// 40 Visualizations/COLLECTOR/VIS_SENSOR_COLLECTOR_TEMP
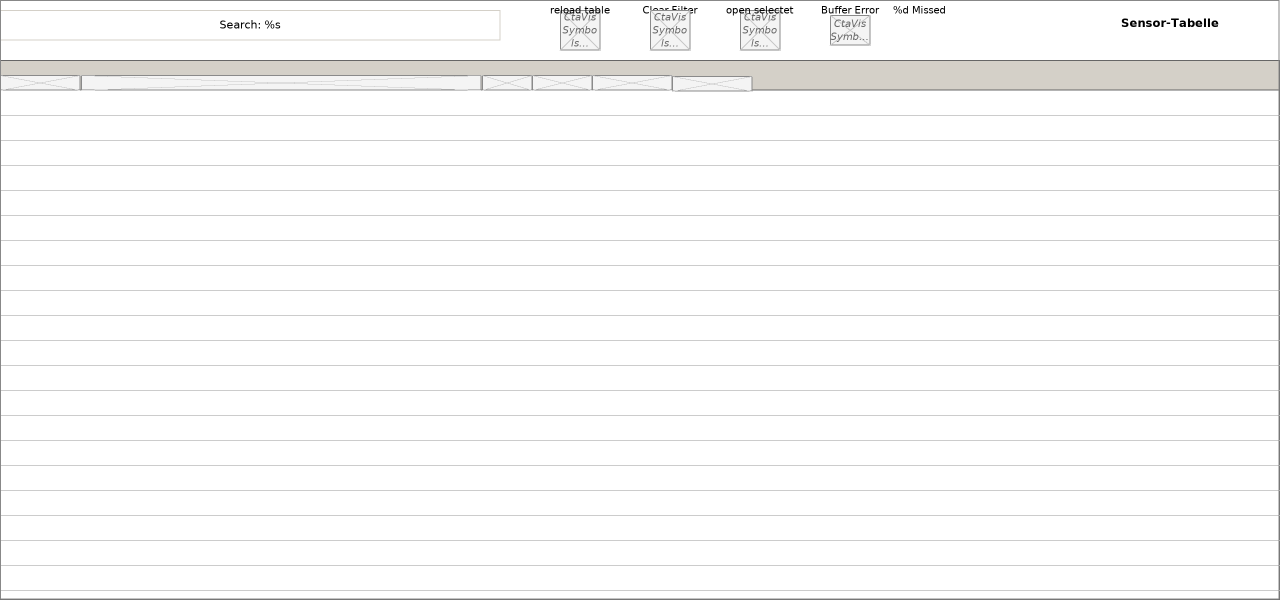
VISUALIZATION VIS_SENSOR_COLLECTOR_TEMP  // 1280x600
VAR_INPUT
	aySensorTabellenInfo   : ARRAY[1..Parameter.iMaxSensor] OF ITF_SENSOR_TABELLE_INFO;
    uiMax                   : UINT;
    ITF_SENSOR_COLLECTOR   : ITF_SENSOR_COLLECTOR;
END_VAR
VAR
    iZeile                  :   INT;
    stSearch                :   STRING;
    uiSort                  :   UINT;
    xReadySearch            :   BOOL;
END_VAR
    Table (0,60 1280x540), data array: aySensorTabellenInfo
        p1128707560: uiMax
        p1014161805: Parameter.iMaxSensor - 1 + 1
        p1137915858: iZeile
        p1933151965: aySensorTabellenInfo[INDEX].proNoBmkInList
        p3863566920: aySensorTabellenInfo[INDEX].proGetInstancePath
        p2192122294: aySensorTabellenInfo[INDEX].proSetInstancePath
        p3854506369: aySensorTabellenInfo[INDEX].proGetBMK
        p516019884: aySensorTabellenInfo[INDEX].proGetObjectId
        p2243050616: aySensorTabellenInfo[INDEX].proGetCustomerDesignation
        p4088588272: aySensorTabellenInfo[INDEX].proGetAKS
        p1892666644: aySensorTabellenInfo[INDEX].proGetVendorDesignation
        p511219082: Vendor designation
        p1757482276: Value OUT
        p746581629: aySensorTabellenInfo[INDEX].proSoftwareValue
        p4092479075: Enabled
        p2170511999: aySensorTabellenInfo[INDEX].proEnSymbol
        p338671338: aySensorTabellenInfo[INDEX].proStateSymbol
        p1218418051: aySensorTabellenInfo[INDEX].proRawValue
        p505689113: Value IN
        p3723444502: aySensorTabellenInfo[INDEX].proPhysicalValue
        p2237128397: Physical IN
    Image (740,10 40x40), invisible if: TO_DINT(iZeile) < LOWER_BOUND(aySensorTabellenInfo,1) OR TO_DINT(iZeile) > UPPER_BOUND(aySensorTabellenInfo,1), image: CtaVisSymbols.ImagePool.Sensor_Black
        OnMouseClick:  Dialog=POPUP_SENSOR, Parameters={uiPopUpGruppe: 0, ITF_SENSORIN: ITF_SENSOR_COLLECTOR.metGetAntriebITF(iZeile)}, OpenModal=True, OpenCentered=True
    Textfield (0,10 500x30), "Search: %s", text variable: stSearch
        OnMouseClick: write the text variable via Default
        OnMouseClick: execute { xReadySearch := TRUE; }
    Image (560,10 40x40), invisible if: NOT xReadySearch, image: CtaVisSymbols.ImagePool.refresh_solo_black
        OnMouseClick: execute { ITF_SENSOR_COLLECTOR.metSortArray(stSearch,uiSort); xReadySearch := FALSE; }
    Label (540,5 80x10), "reload table", invisible if: NOT xReadySearch
    Label (720,5 80x10), "open selectet", invisible if: TO_DINT(iZeile) < LOWER_BOUND(aySensorTabellenInfo,1) OR TO_DINT(iZeile) > UPPER_BOUND(aySensorTabellenInfo,1)
    Label (630,5 80x10), "Clear Filter", invisible if: stSearch = '' AND uiSort = 0
    Image (650,10 40x40), invisible if: stSearch = '' AND uiSort = 0, image: CtaVisSymbols.ImagePool.close_solo_black
        OnMouseClick: execute {
            stSearch := '';
            uiSort   := 0;
            ITF_SENSOR_COLLECTOR.metSortArray(stSearch,uiSort);
            xReadySearch := FALSE;
        }
    Label (1095,8 150x30), "Sensor-Tabelle"
    Label (810,5 80x10), "Buffer Error", invisible if: NOT ITF_SENSOR_COLLECTOR.proBufferError
    Image (830,15 40x30), invisible if: NOT ITF_SENSOR_COLLECTOR.proBufferError, image: CtaVisSymbols.ImagePool.CtaError
    Textfield (890,5 100x10), "%d Missed", text variable: ITF_SENSOR_COLLECTOR.proMissedBuffer, invisible if: NOT ITF_SENSOR_COLLECTOR.proBufferError
    Frame (672,61 80x30)
        shows SelSort(uiSel := uiSort, stSearch := stSearch, ITF_SENSOR_COLLECTOR := ITF_SENSOR_COLLECTOR, uiValue := 6)
    Frame (592,60 80x30)
        shows SelSort(uiSel := uiSort, stSearch := stSearch, ITF_SENSOR_COLLECTOR := ITF_SENSOR_COLLECTOR, uiValue := 5)
    Frame (532,60 60x30)
        shows SelSort(uiSel := uiSort, stSearch := stSearch, ITF_SENSOR_COLLECTOR := ITF_SENSOR_COLLECTOR, uiValue := 4)
    Frame (482,60 50x30)
        shows SelSort(uiSel := uiSort, stSearch := stSearch, ITF_SENSOR_COLLECTOR := ITF_SENSOR_COLLECTOR, uiValue := 3)
    Frame (81,60 400x30)
        shows SelSort(uiSel := uiSort, stSearch := stSearch, ITF_SENSOR_COLLECTOR := ITF_SENSOR_COLLECTOR, uiValue := 2)
    Frame (0,60 80x30)
        shows SelSort(uiSel := uiSort, stSearch := stSearch, ITF_SENSOR_COLLECTOR := ITF_SENSOR_COLLECTOR, uiValue := 1)
END_VISUALIZATION

// 40 Visualizations/COLLECTOR/Help Funktionen/SortPfeil
VISUALIZATION SortPfeil  // 15x15
    Image (0,0 15x15), image: CtaVisSymbols.ImagePool.arrow-down_solo_black
END_VISUALIZATION

// 40 Visualizations/POPUP/POPUP_SENSOR
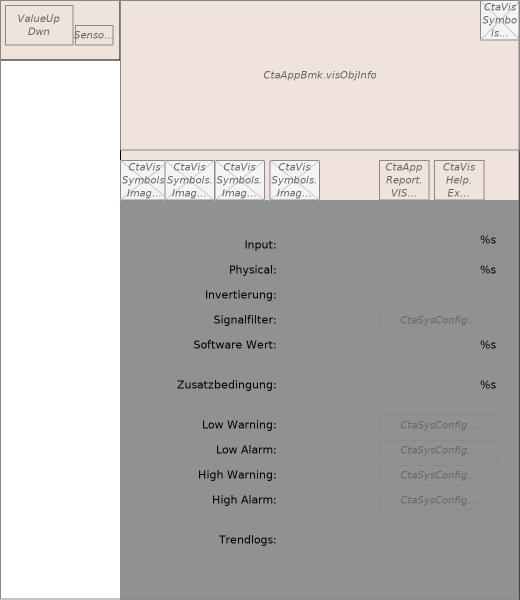
VISUALIZATION POPUP_SENSOR  // 520x600
VAR_INPUT
	ITF_SENSORIN	:	ITF_SENSOR;
	stExklParameter	:	STRING [40];
	uiPopUpGruppe 	: 	UINT;
END_VAR
    Rectangle (0,0 120x60)
    Rectangle (120,0 400x600)
    Frame (120,0 400x150)
        shows CtaAppBmk.visObjInfo(ITF_BMK_IN := ITF_SENSORIN)
    Image (480,0 40x40), image: CtaVisSymbols.ImagePool.close_solo_black
        OnMouseClick:  Dialog=POPUP_SENSOR, Result=None, NumpadKeypadSet=True
    Frame (120,200 399x400), frame switch variable: uiPopUpGruppe
        shows VIS_SENSOR_OVERVIEW(ITF_SENSORIN := ITF_SENSORIN)
        shows VIS_SENSOR_MANUAL(ITF_SENSORIN := ITF_SENSORIN)
        shows VIS_SENSOR_PARAMETER(ITF_SENSORIN := ITF_SENSORIN)
        shows Sensor_BUS(ITF_SENSORIN := ITF_SENSORIN)
        shows VIS_SENSOR_REPORTS(ITF_SENSORIN := ITF_SENSORIN)
        shows VIS_ANTRIEB_REPORTS(ITF_SENSORIN := ITF_SENSOR_IN)
    Frame (120,160 399x40)
        shows VIS_SENSOR_LISTE(uiPopUpGruppe := uiPopUpGruppe, xHand := ITF_SENSORIN.proIsHandOnOrOff, xHandOff := ITF_SENSORIN.proHandOff, ITF_REPORTMANAGER_IN := ITF_SENSORIN.proITF_REPORTMANAGER, stExklParameter := stExklParameter)
        pReferences[0]: AnzError=ITF_SENSORIN.proCountedError, AnzWarning=ITF_SENSORIN.proCountedWarning
    Frame (5,5 110x50), input disabled if: TRUE, frame switch variable: ITF_SENSORIN.proAtIconNr
        shows VIS_SENSOR_FLAT_LEFT_ABOVE(ITF_SENSOR_IN := ITF_SENSORIN, stExklParameter := stExklParameter)
        shows VIS_SENSOR_FLAT_LEFT_BELOW(ITF_SENSOR_IN := ITF_SENSORIN, stExklParameter := stExklParameter)
        shows VIS_SENSOR_FLAT_RIGHT_ABOVE(ITF_SENSOR_IN := ITF_SENSORIN, stExklParameter := stExklParameter)
        shows VIS_SENSOR_FLAT_RIGHT_BELOW(ITF_SENSOR_IN := ITF_SENSORIN, stExklParameter := stExklParameter)
        shows VIS_SENSOR_ROUND_RIGHT_ABOVE(ITF_SENSOR_IN := ITF_SENSORIN, stExklParameter := stExklParameter)
        shows VIS_SENSOR_ROUND_RIGHT_BELOW(ITF_SENSOR_IN := ITF_SENSORIN, stExklParameter := stExklParameter)
        shows VIS_SENSOR_ROUND_LEFT_ABOVE(ITF_SENSOR_IN := ITF_SENSORIN, stExklParameter := stExklParameter)
        shows VIS_SENSOR_ROUND_LEFT_BELOW(ITF_SENSOR_IN := ITF_SENSORIN, stExklParameter := stExklParameter)
END_VISUALIZATION

// 40 Visualizations/POPUP/VIS_SENSOR_LISTE
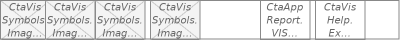
VISUALIZATION VIS_SENSOR_LISTE  // 400x40
VAR_IN_OUT
	uiPopUpGruppe : UINT;
END_VAR
VAR_INPUT
    xHand           		: BOOL;
    xHandOff        		: BOOL;
    ITF_REPORTMANAGER_IN    : CtaAppReport.ITF_REPORTMANAGER;
	stExklParameter			: STRING [40];
END_VAR
    Rectangle (5,0 40x40), colour toggle: uiPopUpGruppe = 0
        OnMouseDown: execute { uiPopUpGruppe := 0; }
    Image (0,0 50x40), image: CtaVisSymbols.ImagePool.eye
        OnMouseDown: execute { uiPopUpGruppe := 0; }
    Rectangle (50,0 40x40), colour toggle: uiPopUpGruppe = 1
        OnMouseDown: execute { uiPopUpGruppe := 1; }
    Image (45,0 50x40), invisible if: NOT xHand, image: CtaVisSymbols.ImagePool.front_hand_Yellow
        OnMouseDown: execute { uiPopUpGruppe := 1; }
    Image (45,0 50x40), image: CtaVisSymbols.ImagePool.front_hand_Black
        OnMouseDown: execute { uiPopUpGruppe := 1; }
    Image (45,0 50x40), invisible if: NOT xHandOff, image: CtaVisSymbols.ImagePool.front_hand_Yellow_Off
        OnMouseDown: execute { uiPopUpGruppe := 1; }
    Rectangle (100,0 40x40), colour toggle: uiPopUpGruppe = 2
        OnMouseDown: execute { uiPopUpGruppe := 2; }
    Image (95,0 50x40), image: CtaVisSymbols.ImagePool.gear
        OnMouseDown: execute { uiPopUpGruppe := 2; }
    Rectangle (155,0 40x40), colour toggle: uiPopUpGruppe = 3
        OnMouseDown: execute { uiPopUpGruppe := 3; }
    Image (150,0 50x40), image: CtaVisSymbols.ImagePool.lan
        OnMouseDown: execute { uiPopUpGruppe := 3; }
    Rectangle (265,0 40x40), colour toggle: uiPopUpGruppe = 4
        OnMouseDown: execute { uiPopUpGruppe := 4; }
    Frame (260,0 50x40)
        shows CtaAppReport.VIS_ANZ_REPORTS_MODUL(ITF_REPORTMANAGER_IN := ITF_REPORTMANAGER_IN)
        OnMouseClick: execute { uiPopUpGruppe := 4; }
    Rectangle (320,0 40x40)
    Frame (315,0 50x40)
        shows CtaVisHelp.ExkParameterSymbol(stExklParameter := stExklParameter)
END_VISUALIZATION

// 40 Visualizations/POPUP/PARAMETER/SENSOR_ReportManagement/Sensor_LowAlarm_Param
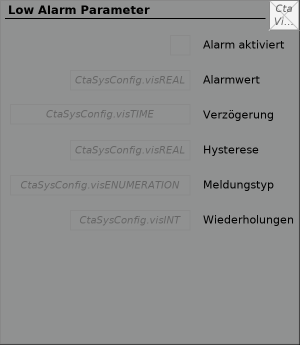
VISUALIZATION Sensor_LowAlarm_Param  // 300x345
VAR_INPUT
	ITF_SENSORIN	:	ITF_SENSOR;
END_VAR
VAR_IN_OUT
    xShow   :   BOOL;
END_VAR
    Rectangle (0,0 300x345)
    Image (269,0 30x30), image: CtaVisSymbols.ImagePool.close_solo_black
        OnMouseClick: execute { xShow := FALSE; }
    Label (5,0 198x20), "Low Alarm Parameter"
    Line (5,18) (265,18)
    Label (200,35 100x20), "Alarm aktiviert"
    Frame (170,35 20x20)
        shows CtaSysConfig.visBOOL(visfbBOOLIn := ITF_SENSORIN.P_scLoAlarm_fbxDoesAlarm)
    Label (200,70 100x20), "Alarmwert"
    Frame (70,70 120x20), invisible if: (ITF_SENSORIN.proValueInputType = enInputType.DigitalInput) OR (ITF_SENSORIN.proValueInputType = enInputType.Digital_ITF_Input)
        shows CtaSysConfig.visREAL(visfbREALIn := ITF_SENSORIN.P_scLoAlarm_fbrValue)
    Label (200,105 100x20), "Verzögerung"
    Frame (10,104 180x20)
        shows CtaSysConfig.visTIME(visfbTIMEIn := ITF_SENSORIN.P_scLoAlarm_fbtDelayTillAlarm)
    Frame (70,140 120x20), invisible if: (ITF_SENSORIN.proValueInputType = enInputType.DigitalInput) OR (ITF_SENSORIN.proValueInputType = enInputType.Digital_ITF_Input)
        shows CtaSysConfig.visREAL(visfbREALIn := ITF_SENSORIN.P_scLoAlarm_fbrHysterese)
    Label (200,140 100x20), "Hysterese"
    Frame (10,175 180x20), text list: 'CtaAppReport.txtLibAp99_2enTypeOfAck', text index: CtaSysConfig.fcGetEnumerationId(ITF_SENSORIN.P_scLoAlarm_fbiTypeOfAcknolage)
        shows CtaSysConfig.visENUMERATION(visfbENUIn := ITF_SENSORIN.P_scLoAlarm_fbiTypeOfAcknolage)
    Label (200,175 100x20), "Meldungstyp"
    Frame (70,210 120x20), invisible if: NOT (CtaSysConfig.fcGetEnumerationId(ITF_SENSORIN.P_scLoAlarm_fbiTypeOfAcknolage) = 2)
        shows CtaSysConfig.visINT(visfbINTIn := ITF_SENSORIN.P_scLoAlarm_fbiRetryTillLock)
    Label (200,210 100x20), "Wiederholungen"
END_VISUALIZATION

// 40 Visualizations/ICON/SENSOR_FLAT/SENSOR_FLAT_TXT_LEFT/ABOVE/VIS_SENSOR_FLAT_LeftAboveCheckQuerry
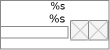
VISUALIZATION VIS_SENSOR_FLAT_LeftAboveCheckQuerry  // 110x50
VAR_INPUT
    ITF_SENSOR_IN   :   ITF_SENSOR;
	stExklParameter	:	STRING [40];	
END_VAR
    Frame (0,0 110x50)
        shows VIS_SENSOR_FLAT_LeftAboveCheckIsEnabled(ITF_SENSOR_IN := ITF_SENSOR_IN, stExklParameter := stExklParameter)
END_VISUALIZATION

// 40 Visualizations/ICON/SENSOR_FLAT/SENSOR_FLAT_TXT_LEFT/ABOVE/VIS_SENSOR_FLAT_LEFT_ABOVE
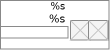
VISUALIZATION VIS_SENSOR_FLAT_LEFT_ABOVE  // 110x50
VAR_INPUT
    ITF_SENSOR_IN   :   ITF_SENSOR;	
END_VAR
VAR_INPUT CONSTANT	
	stExklParameter	:	STRING [40] := ' ';	
END_VAR
VAR CONSTANT
	uiIconNr		: UINT := 0;
END_VAR
    Frame (0,0 110x50), invisible if: NOT fcCheckQuerryAndIconReturn(_ITF_IN := ITF_SENSOR_IN, _uiIconNr_IN := uiIconNr)
        shows VIS_SENSOR_FLAT_LeftAboveCheckQuerry(ITF_SENSOR_IN := ITF_SENSOR_IN, stExklParameter := stExklParameter)
END_VISUALIZATION

// 40 Visualizations/ICON/SENSOR_FLAT/SENSOR_FLAT_TXT_LEFT/ABOVE/VIS_SENSOR_FLAT_LeftAboveCheckIsEnabled
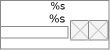
VISUALIZATION VIS_SENSOR_FLAT_LeftAboveCheckIsEnabled  // 110x50
VAR_INPUT
    ITF_SENSOR_IN   :   ITF_SENSOR;
	stExklParameter	:	STRING [40];	
END_VAR
    Frame (70,20 38x20), invisible if: NOT ITF_SENSOR_IN.proIsEnabled
        shows SensorFlat(ITF_SENSORIN := ITF_SENSOR_IN)
    Frame (0,0 68x40), invisible if: NOT ITF_SENSOR_IN.proIsEnabled
        shows ValueUpDwn(ITF_SENSORIN := ITF_SENSOR_IN, uiTextAusrichtung := 6)
    Rectangle (0,0 110x50)
        OnMouseClick:  Dialog=POPUP_SENSOR, Parameters={stExklParameter: stExklParameter, ITF_SENSORIN: ITF_SENSOR_IN, uiPopUpGruppe: 0}, OpenCentered=True
END_VISUALIZATION

// 40 Visualizations/ICON/SENSOR_FLAT/SENSOR_FLAT_TXT_RIGHT/ABOVE/VIS_SENSOR_FLAT_RigthAboveCheckIsEnabled
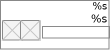
VISUALIZATION VIS_SENSOR_FLAT_RigthAboveCheckIsEnabled  // 110x50
VAR_INPUT
    ITF_SENSOR_IN   :   ITF_SENSOR;
	stExklParameter	:	STRING [40];	
END_VAR
    Frame (2,20 38x20), invisible if: NOT ITF_SENSOR_IN.proIsEnabled
        shows SensorFlat(ITF_SENSORIN := ITF_SENSOR_IN)
    Frame (42,0 68x40), invisible if: NOT ITF_SENSOR_IN.proIsEnabled
        shows ValueUpDwn(ITF_SENSORIN := ITF_SENSOR_IN, uiTextAusrichtung := 4)
    Rectangle (0,0 110x50)
        OnMouseClick:  Dialog=POPUP_SENSOR, Parameters={stExklParameter: stExklParameter, ITF_SENSORIN: ITF_SENSOR_IN, uiPopUpGruppe: 0}, OpenCentered=True
END_VISUALIZATION

// 40 Visualizations/ICON/SENSOR_BASE/ICON/Flat/SensorFlat
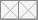
VISUALIZATION SensorFlat  // 38x20
VAR_INPUT
    ITF_SENSORIN   :   ITF_SENSOR;	
END_VAR
    RoundedRectangle (0,0 38x20), colour toggle: ITF_SENSORIN.proAcknowlege, invisible if: ITF_SENSORIN.proIsError
    RoundedRectangle (0,0 38x20), colour toggle: ITF_SENSORIN.proIsError
    Image (0,0 20x20), invisible if: NOT ITF_SENSORIN.proIsWarning, image: CtaVisSymbols.ImagePool.CtaWarning
    Image (18,0 20x20), invisible if: NOT ITF_SENSORIN.proIsHandOnOrOff, image: CtaVisSymbols.ImagePool.front_hand_Yellow
    Image (18,0 20x20), invisible if: NOT ITF_SENSORIN.proHandOff, image: CtaVisSymbols.ImagePool.front_hand_Yellow_Off
END_VISUALIZATION

// 40 Visualizations/POPUP/PARAMETER/VIS_SENSOR_PARAMETER
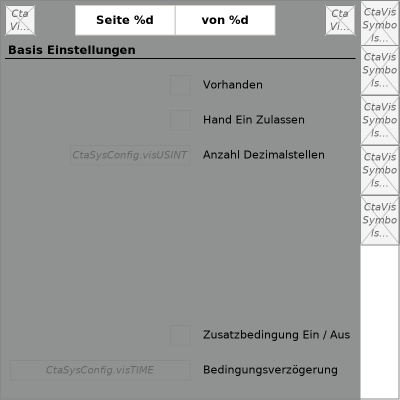
VISUALIZATION VIS_SENSOR_PARAMETER  // 400x400
VAR_INPUT
    ITF_SENSORIN : ITF_SENSOR;
END_VAR
VAR
    uiParameterGruppe : UINT;
END_VAR
    Image (145,122 150x30), image: ImagePool.Kreis
    Frame (360,0 40x300)
        shows VIS_SENSOR_PARAMETER_LISTE(enValueInputType := ITF_SENSORIN.proValueInputType, uiParameterGruppe := uiParameterGruppe)
    Frame (0,0 360x400), frame switch variable: uiParameterGruppe
        shows VIS_SENSOR_PARAMETER_BASE(ITF_SENSORIN := ITF_SENSORIN)
        shows VIS_SENSOR_PARAMETER_FILTER(ITF_SENSORIN := ITF_SENSORIN)
        shows VIS_SENSOR_PARAMETER_REPORTMNG(ITF_SENSORIN := ITF_SENSORIN)
        shows VIS_SENSOR_IO_PARAMETER(ITF_SENSORIN := ITF_SENSORIN)
        shows VIS_SENSOR_PARAMETER_TRENDLOG(ITF_SENSORIN := ITF_SENSORIN)
        pReferences[3]: ITF_IO_IN=ITF_SENSOR_IN.proIO_ITF
END_VISUALIZATION

// 40 Visualizations/POPUP/PARAMETER/VIS_SENSOR_PARAMETER_LISTE
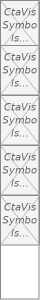
VISUALIZATION VIS_SENSOR_PARAMETER_LISTE  // 40x300
VAR_INPUT
	enValueInputType : enInputType;
END_VAR
VAR_IN_OUT
	uiParameterGruppe : UINT;
END_VAR
    Rectangle (0,5 39x40), colour toggle: uiParameterGruppe = 0
        OnMouseDown: execute { uiParameterGruppe := 0; }
    Image (0,0 40x50), image: CtaVisSymbols.ImagePool.Sensor_Black
        OnMouseDown: execute { uiParameterGruppe := 0; }
    Rectangle (0,50 39x40), colour toggle: uiParameterGruppe = 1
        OnMouseDown: execute { uiParameterGruppe := 1; }
    Image (0,45 40x50), image: CtaVisSymbols.ImagePool.SearchFilter
        OnMouseDown: execute { uiParameterGruppe := 1; }
    Rectangle (0,100 39x40), colour toggle: uiParameterGruppe = 2
        OnMouseDown: execute { uiParameterGruppe := 2; }
    Image (0,95 40x50), image: CtaVisSymbols.ImagePool.notification_black
        OnMouseDown: execute { uiParameterGruppe := 2; }
    Rectangle (1,150 39x40), colour toggle: uiParameterGruppe = 3, invisible if: enValueInputType = 0 OR enValueInputType = 1 OR enValueInputType = 2, input disabled if: enValueInputType = 0 OR enValueInputType = 1 OR enValueInputType = 2
        OnMouseDown: execute { uiParameterGruppe := 3; }
    Image (0,145 40x50), invisible if: enValueInputType = 0 OR enValueInputType = 1 OR enValueInputType = 2, input disabled if: enValueInputType = 0 OR enValueInputType = 1 OR enValueInputType = 2, image: CtaVisSymbols.ImagePool.dip-switch
        OnMouseDown: execute { uiParameterGruppe := 3; }
    Rectangle (0,200 39x40), colour toggle: uiParameterGruppe = 4
        OnMouseDown: execute { uiParameterGruppe := 4; }
    Image (0,195 40x50), image: CtaVisSymbols.ImagePool.sine-wave
        OnMouseDown: execute { uiParameterGruppe := 4; }
END_VISUALIZATION

// 40 Visualizations/POPUP/MANUAL/VIS_SENSOR_MANUAL
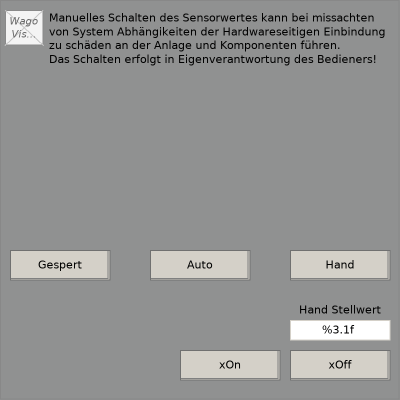
VISUALIZATION VIS_SENSOR_MANUAL  // 400x400
VAR_INPUT
    ITF_SENSORIN    :   ITF_SENSOR;	
END_VAR
    Button (10,250 100x30), "Gespert", colour toggle: ITF_SENSORIN.proHandOff, pressed state: ITF_SENSORIN.proHandOff
        toggle ITF_SENSORIN.proHandOff
    Button (290,250 100x30), "Hand", colour toggle: ITF_SENSORIN.proHandOn, pressed state: ITF_SENSORIN.proHandOn
        toggle ITF_SENSORIN.proHandOn
    Button (150,250 100x30), "Auto", colour toggle: ITF_SENSORIN.proAuto, pressed state: ITF_SENSORIN.proAuto
        toggle ITF_SENSORIN.proAuto
    Label (46,10 350x100), "Manuelles Schalten des Sensorwertes kann bei missachten von System Abhängikeiten der Hardwareseitigen Einbindung zu schäden an der Anlage und Komponenten führen. Das Schalten erfolgt in Eigenverantwortung des Bedieners!"
    Textfield (290,320 100x20), "%3.1f", text variable: ITF_SENSORIN.proHandOnY, invisible if: ITF_SENSORIN.proValueInputType = 0 OR ITF_SENSORIN.proValueInputType = 2 OR ITF_SENSORIN.proValueInputType = 4
        OnMouseClick: write the text variable via InputWithLimits, min 0, max 100, title 'Stellwert'
    Image (5,10 38x35), image: WagoVisuIcons.WagoIcons.2
    Label (290,300 100x20), "Hand Stellwert"
    Button (290,350 100x30), "xOff", colour toggle: ITF_SENSORIN.proManualFalse, pressed state: ITF_SENSORIN.proManualFalse, invisible if: ITF_SENSORIN.proValueInputType = 0 OR ITF_SENSORIN.proValueInputType = 1 OR ITF_SENSORIN.proValueInputType = 3
        toggle ITF_SENSORIN.proManualFalse
    Button (180,350 100x30), "xOn", colour toggle: ITF_SENSORIN.proManualTrue, pressed state: ITF_SENSORIN.proManualTrue, invisible if: ITF_SENSORIN.proValueInputType = 0 OR ITF_SENSORIN.proValueInputType = 1 OR ITF_SENSORIN.proValueInputType = 3
        toggle ITF_SENSORIN.proManualTrue
END_VISUALIZATION

// 40 Visualizations/POPUP/OVERVIEW/VIS_SENSOR_OVERVIEW
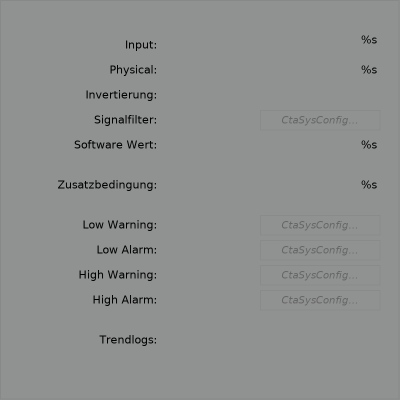
VISUALIZATION VIS_SENSOR_OVERVIEW  // 400x400
VAR_INPUT
    ITF_SENSORIN	:	ITF_SENSOR;
END_VAR
    Frame (0,0 400x400), invisible if: NOT __QUERYINTERFACE(ITF_SENSORIN,ITF_SENSORIN)
        shows VIS_SENSOR_OVERVIEW0(ITF_SENSORIN := ITF_SENSORIN)
END_VISUALIZATION

// 40 Visualizations/POPUP/PARAMETER/SENSOR_ReportManagement/Sensor_HighAlarm_Param
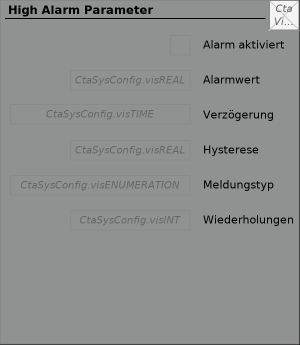
VISUALIZATION Sensor_HighAlarm_Param  // 300x345
VAR_INPUT
	ITF_SENSORIN	:	ITF_SENSOR;
END_VAR
VAR_IN_OUT
    xShow   :   BOOL;
END_VAR
    Rectangle (0,0 300x345)
    Image (269,0 30x30), image: CtaVisSymbols.ImagePool.close_solo_black
        OnMouseClick: execute { xShow := FALSE; }
    Label (5,0 198x20), "High Alarm Parameter"
    Line (5,18) (265,18)
    Label (200,35 100x20), "Alarm aktiviert"
    Frame (170,35 20x20)
        shows CtaSysConfig.visBOOL(visfbBOOLIn := ITF_SENSORIN.P_scHighAlram_fbxDoesAlarm)
    Label (200,70 100x20), "Alarmwert"
    Frame (70,70 120x20), invisible if: (ITF_SENSORIN.proValueInputType = enInputType.DigitalInput) OR (ITF_SENSORIN.proValueInputType = enInputType.Digital_ITF_Input)
        shows CtaSysConfig.visREAL(visfbREALIn := ITF_SENSORIN.P_scHighAlarm_fbrValue)
    Label (200,105 100x20), "Verzögerung"
    Frame (10,104 180x20)
        shows CtaSysConfig.visTIME(visfbTIMEIn := ITF_SENSORIN.P_scHighAlarm_fbtDelayTillAlarm)
    Frame (70,140 120x20), invisible if: (ITF_SENSORIN.proValueInputType = enInputType.DigitalInput) OR (ITF_SENSORIN.proValueInputType = enInputType.Digital_ITF_Input)
        shows CtaSysConfig.visREAL(visfbREALIn := ITF_SENSORIN.P_scHighAlarm_fbrHysterese)
    Label (200,140 100x20), "Hysterese"
    Frame (10,175 180x20), text list: 'CtaAppReport.txtLibAp99_2enTypeOfAck', text index: CtaSysConfig.fcGetEnumerationId(ITF_SENSORIN.P_scHighAlarm_fbiTypeOfAcknolage)
        shows CtaSysConfig.visENUMERATION(visfbENUIn := ITF_SENSORIN.P_scHighAlarm_fbiTypeOfAcknolage)
    Label (200,175 100x20), "Meldungstyp"
    Frame (70,210 120x20), invisible if: NOT (CtaSysConfig.fcGetEnumerationId(ITF_SENSORIN.P_scHighAlarm_fbiTypeOfAcknolage) = 2)
        shows CtaSysConfig.visINT(visfbINTIn := ITF_SENSORIN.P_scHighAlarm_fbiRetryTillLock)
    Label (200,210 100x20), "Wiederholungen"
END_VISUALIZATION

// 40 Visualizations/ICON/SENSOR_FLAT/SENSOR_FLAT_TXT_LEFT/BELOW/VIS_SENSOR_FLAT_LEFT_BELOW
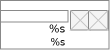
VISUALIZATION VIS_SENSOR_FLAT_LEFT_BELOW  // 110x50
VAR_INPUT
    ITF_SENSOR_IN   :   ITF_SENSOR;	
END_VAR
VAR_INPUT CONSTANT	
	stExklParameter	:	STRING [40] := ' ';	
END_VAR
VAR CONSTANT
	uiIconNr		: UINT := 1;
END_VAR
    Frame (0,0 110x50), invisible if: NOT fcCheckQuerryAndIconReturn(_ITF_IN := ITF_SENSOR_IN, _uiIconNr_IN := uiIconNr)
        shows VIS_SENSOR_FLAT_LeftBelowCheckQuerry(ITF_SENSOR_IN := ITF_SENSOR_IN, stExklParameter := stExklParameter)
END_VISUALIZATION

// 40 Visualizations/POPUP/PARAMETER/SENSOR_ReportManagement/Sensor_HighWarning_Param
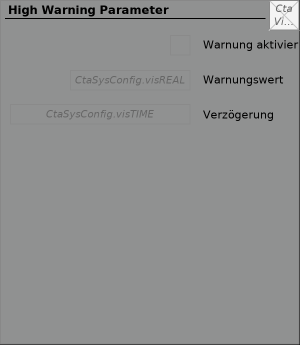
VISUALIZATION Sensor_HighWarning_Param  // 300x345
VAR_INPUT
	ITF_SENSORIN	:	ITF_SENSOR;
END_VAR
VAR_IN_OUT
    xShow   :   BOOL;
END_VAR
    Rectangle (0,0 300x345)
    Image (269,0 30x30), image: CtaVisSymbols.ImagePool.close_solo_black
        OnMouseClick: execute { xShow := FALSE; }
    Label (5,0 198x20), "High Warning Parameter"
    Line (5,18) (265,18)
    Label (200,35 100x20), "Warnung aktiviert"
    Frame (170,35 20x20)
        shows CtaSysConfig.visBOOL(visfbBOOLIn := ITF_SENSORIN.P_scHighWarning_fbxDoesWarning)
    Label (200,70 100x20), "Warnungswert"
    Frame (70,70 120x20), invisible if: (ITF_SENSORIN.proValueInputType = enInputType.DigitalInput) OR (ITF_SENSORIN.proValueInputType = enInputType.Digital_ITF_Input)
        shows CtaSysConfig.visREAL(visfbREALIn := ITF_SENSORIN.P_scHighWarning_fbrValue)
    Label (200,105 100x20), "Verzögerung"
    Frame (10,104 180x20)
        shows CtaSysConfig.visTIME(visfbTIMEIn := ITF_SENSORIN.P_scHighWarning_fbtDelayTillWarning)
END_VISUALIZATION

// 40 Visualizations/ICON/SENSOR_FLAT/SENSOR_FLAT_TXT_LEFT/BELOW/VIS_SENSOR_FLAT_LeftBelowCheckIsEnabled
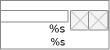
VISUALIZATION VIS_SENSOR_FLAT_LeftBelowCheckIsEnabled  // 110x50
VAR_INPUT
    ITF_SENSOR_IN   :   ITF_SENSOR;
	stExklParameter	:	STRING [40];	
END_VAR
    Frame (70,10 38x20), invisible if: NOT ITF_SENSOR_IN.proIsEnabled
        shows SensorFlat(ITF_SENSORIN := ITF_SENSOR_IN)
    Frame (0,10 68x40), invisible if: NOT ITF_SENSOR_IN.proIsEnabled
        shows ValueDwnUp(ITF_SENSORIN := ITF_SENSOR_IN, uiTextAusrichtung := 6)
    Rectangle (0,0 110x50)
        OnMouseClick:  Dialog=POPUP_SENSOR, Parameters={stExklParameter: stExklParameter, ITF_SENSORIN: ITF_SENSOR_IN, uiPopUpGruppe: 0}, OpenCentered=True
END_VISUALIZATION

// 40 Visualizations/POPUP/REPORTS/VIS_SENSOR_REPORTS
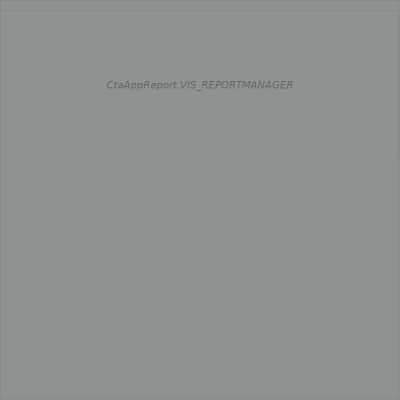
VISUALIZATION VIS_SENSOR_REPORTS  // 400x400
VAR_INPUT
    ITF_SENSORIN    :   ITF_SENSOR;	
END_VAR
    Frame (0,10 400x150)
        shows CtaAppReport.VIS_REPORTMANAGER(ITF_REPORTMANAGER := ITF_SENSORIN.proITF_REPORTMANAGER)
END_VISUALIZATION

// 40 Visualizations/POPUP/PARAMETER/SENSOR_ParameterBase/VIS_SENSOR_PARAMETER_BASE0
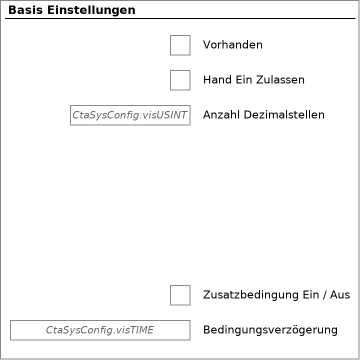
VISUALIZATION VIS_SENSOR_PARAMETER_BASE0  // 360x360
VAR_INPUT
    ITF_SENSORIN	:  ITF_SENSOR;
END_VAR
    Label (5,0 350x20), "Basis Einstellungen"
    Line (5,18) (355,18)
    Label (200,35 150x20), "Vorhanden"
    Label (200,70 150x20), "Hand Ein Zulassen"
    Frame (170,35 20x20)
        shows CtaSysConfig.visBOOL(visfbBOOLIn := ITF_SENSORIN.P_scBase_fbxEnable)
    Frame (170,70 20x20)
        shows CtaSysConfig.visBOOL(visfbBOOLIn := ITF_SENSORIN.P_scManual_fbxAllowManualOn)
    Frame (170,285 20x20)
        shows CtaSysConfig.visBOOL(visfbBOOLIn := ITF_SENSORIN.P_scAlCondition_fbxEnable)
    Label (200,285 150x20), "Zusatzbedingung Ein / Aus"
    Frame (10,320 180x20)
        shows CtaSysConfig.visTIME(visfbTIMEIn := ITF_SENSORIN.P_scAlCondition_fbtDelayTillCondition)
    Label (200,320 150x20), "Bedingungsverzögerung"
    Frame (70,105 120x20), invisible if: NOT (ITF_SENSORIN.proValueInputType = enInputType.AnalogInput or ITF_SENSORIN.proValueInputType = enInputType.Analog_ITF_Input)
        shows CtaSysConfig.visUSINT(visfbUSINTIn := ITF_SENSORIN.P_scVisu_fbusiDezimalPos)
    Label (200,105 150x20), "Anzahl Dezimalstellen", invisible if: NOT (ITF_SENSORIN.proValueInputType = enInputType.AnalogInput or ITF_SENSORIN.proValueInputType = enInputType.Analog_ITF_Input)
END_VISUALIZATION

// 40 Visualizations/POPUP/PARAMETER/SENSOR_ParameterBase/VIS_SENSOR_PARAMETER_BASE
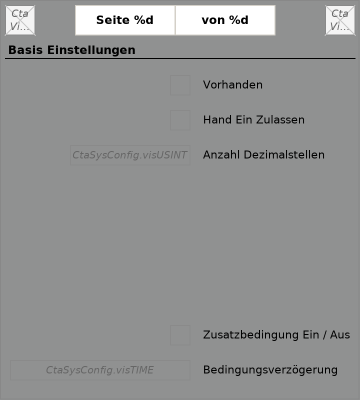
VISUALIZATION VIS_SENSOR_PARAMETER_BASE  // 360x400
VAR_INPUT
    ITF_SENSORIN 	: 	ITF_SENSOR;
END_VAR
VAR
    uiPage  :   UINT;
    uiMin   :   UINT    := 0;
    uiMax   :   UINT    := 0;
END_VAR
    Image (5,5 30x30), invisible if: uiPage = uiMin, image: CtaVisSymbols.ImagePool.arrow-left_square
        OnMouseClick: execute {
            uiPage := uiPage - 1;
            IF uiPage <= uiMin THEN
                uiPage := uiMin;
            END_IF;
        }
    Image (325,5 30x30), invisible if: uiPage = uiMax, image: CtaVisSymbols.ImagePool.arrow-right_square
        OnMouseClick: execute {
            uiPage := uiPage + 1;
            IF uiPage >= uiMax THEN
                uiPage := uiMax;
            END_IF;
        }
    Frame (0,40 360x360), frame switch variable: uiPage
        shows VIS_SENSOR_PARAMETER_BASE0(ITF_SENSORIN := ITF_SENSORIN)
        shows AT_ParameterIO1(ITF_Parameter := ITF_Parameter)
        pReferences[0]: ITF_Parameter=ITF_Parameter
    Textfield (175,5 100x30), "von %d", text variable: uiMax
    Textfield (75,5 100x30), "Seite %d", text variable: uiPage
END_VISUALIZATION

// 40 Visualizations/ICON/SENSOR_FLAT/SENSOR_FLAT_TXT_RIGHT/ABOVE/VIS_SENSOR_FLAT_RIGHT_ABOVE
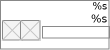
VISUALIZATION VIS_SENSOR_FLAT_RIGHT_ABOVE  // 110x50
VAR_INPUT
    ITF_SENSOR_IN   :   ITF_SENSOR;	
END_VAR
VAR_INPUT CONSTANT	
	stExklParameter	:	STRING [40] := ' ';	
END_VAR
VAR CONSTANT
	uiIconNr		:	UINT := 2;
END_VAR
    Frame (0,0 110x50), invisible if: NOT fcCheckQuerryAndIconReturn(_ITF_IN := ITF_SENSOR_IN, _uiIconNr_IN := uiIconNr)
        shows VIS_SENSOR_FLAT_RigthAboveCheckQuerry(ITF_SENSOR_IN := ITF_SENSOR_IN, stExklParameter := stExklParameter)
END_VISUALIZATION

// 40 Visualizations/ICON/SENSOR_FLAT/SENSOR_FLAT_TXT_LEFT/BELOW/VIS_SENSOR_FLAT_LeftBelowCheckQuerry
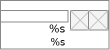
VISUALIZATION VIS_SENSOR_FLAT_LeftBelowCheckQuerry  // 110x50
VAR_INPUT
    ITF_SENSOR_IN   :   ITF_SENSOR;
	stExklParameter	:	STRING [40];	
END_VAR
    Frame (0,0 110x50)
        shows VIS_SENSOR_FLAT_LeftBelowCheckIsEnabled(ITF_SENSOR_IN := ITF_SENSOR_IN, stExklParameter := stExklParameter)
END_VISUALIZATION

// 40 Visualizations/POPUP/PARAMETER/SENSOR_ReportManagement/VIS_SENSOR_PARAMETER_REPORTMNG
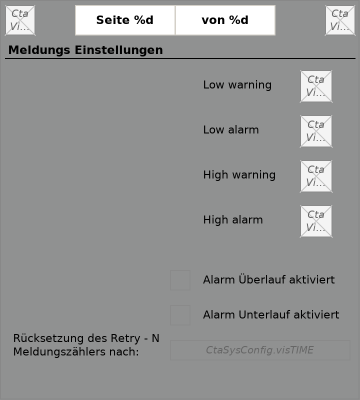
VISUALIZATION VIS_SENSOR_PARAMETER_REPORTMNG  // 360x400
VAR_INPUT
   	ITF_SENSORIN	:	ITF_SENSOR;
END_VAR
VAR
    uiPage  :   UINT;
    uiMin   :   UINT    := 0;
    uiMax   :   UINT    := 0;
END_VAR
    Image (5,5 30x30), invisible if: uiPage = uiMin, image: CtaVisSymbols.ImagePool.arrow-left_square
        OnMouseClick: execute {
            uiPage := uiPage - 1;
            IF uiPage <= uiMin THEN
                uiPage := uiMin;
            END_IF;
        }
    Image (325,5 30x30), invisible if: uiPage = uiMax, image: CtaVisSymbols.ImagePool.arrow-right_square
        OnMouseClick: execute {
            uiPage := uiPage + 1;
            IF uiPage >= uiMax THEN
                uiPage := uiMax;
            END_IF;
        }
    Frame (0,40 360x360), frame switch variable: uiPage
        shows VIS_SENSOR_PARAMETER_REPORTMNG_1(ITF_SENSORIN := ITF_SENSORIN)
        shows AT_ParameterIO1(ITF_Parameter := ITF_Parameter)
    Textfield (175,5 100x30), "von %d", text variable: uiMax
    Textfield (75,5 100x30), "Seite %d", text variable: uiPage
END_VISUALIZATION

// 40 Visualizations/POPUP/PARAMETER/SENSOR_ReportManagement/VIS_SENSOR_PARAMETER_REPORTMNG_1
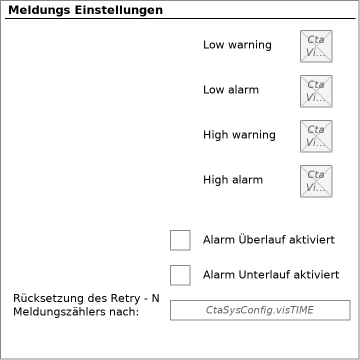
VISUALIZATION VIS_SENSOR_PARAMETER_REPORTMNG_1  // 360x360
VAR_INPUT
   	ITF_SENSORIN	:	ITF_SENSOR;
END_VAR
VAR
	xShowLoWarning	:	BOOL;
	xShowLoAlarm	:	BOOL;
	xShowHiWarning	:	BOOL;
	xShowHiAlarm	:	BOOL;
END_VAR
    Label (5,0 350x20), "Meldungs Einstellungen"
    Line (5,18) (355,18)
    Label (200,35 150x20), "Low warning"
    Label (200,80 150x20), "Low alarm"
    Label (200,125 150x20), "High warning"
    Label (200,170 150x20), "High alarm"
    Image (300,30 32x32), image: CtaVisSymbols. ImagePool.CtaInfo
        OnMouseClick: execute {
            xShowLoWarning	:=	TRUE;
            xShowLoAlarm	:=	FALSE;
            xShowHiWarning	:=	FALSE;
            xShowHiAlarm	:=	FALSE;
        }
    Frame (400,18 300x345), invisible if: NOT xShowLoWarning
        shows Sensor_LowWarning_Param(ITF_SENSORIN := ITF_SENSORIN, xShow := xShowLoWarning)
    Image (300,75 32x32), image: CtaVisSymbols.ImagePool.CtaInfo
        OnMouseClick: execute {
            xShowLoWarning	:=	FALSE;
            xShowLoAlarm	:=	TRUE;
            xShowHiWarning	:=	FALSE;
            xShowHiAlarm	:=	FALSE;
        }
    Frame (400,18 300x345), invisible if: NOT xShowLoAlarm
        shows Sensor_LowAlarm_Param(ITF_SENSORIN := ITF_SENSORIN, xShow := xShowLoAlarm)
    Image (300,120 32x32), image: CtaVisSymbols.ImagePool.CtaInfo
        OnMouseClick: execute {
            xShowLoWarning	:=	FALSE;
            xShowLoAlarm	:=	FALSE;
            xShowHiWarning	:=	TRUE;
            xShowHiAlarm	:=	FALSE;
        }
    Frame (400,18 300x345), invisible if: NOT xShowHiWarning
        shows Sensor_HighWarning_Param(ITF_SENSORIN := ITF_SENSORIN, xShow := xShowHiWarning)
    Image (300,165 32x32), image: CtaVisSymbols.ImagePool.CtaInfo
        OnMouseClick: execute {
            xShowLoWarning	:=	FALSE;
            xShowLoAlarm	:=	FALSE;
            xShowHiWarning	:=	FALSE;
            xShowHiAlarm	:=	TRUE;
        }
    Frame (400,18 300x345), invisible if: NOT xShowHiAlarm
        shows Sensor_HighAlarm_Param(ITF_SENSORIN := ITF_SENSORIN, xShow := xShowHiAlarm)
    Frame (170,230 20x20)
        shows CtaSysConfig.visBOOL(visfbBOOLIn := ITF_SENSORIN.P_scAnalogAlarm_fbxEnableOverflowAl)
    Label (200,230 160x20), "Alarm Überlauf aktiviert"
    Label (200,265 160x20), "Alarm Unterlauf aktiviert"
    Frame (170,265 20x20)
        shows CtaSysConfig.visBOOL(visfbBOOLIn := ITF_SENSORIN.P_scAnalogAlarm_fbxEnableUnderflowAl)
    Frame (170,300 180x20)
        shows CtaSysConfig.visTIME(visfbTIMEIn := ITF_SENSORIN.P_scAlarmReset_fbtDealyTillReset)
    Label (10,285 160x40), "Rücksetzung des Retry - N Meldungszählers nach:"
END_VISUALIZATION

// 40 Visualizations/POPUP/PARAMETER/SENSOR_Filter/VIS_SENSOR_PARAMETER_FILTER
